PROGRAM MAIN
VAR
	//Required functions
	fbJson:FB_JsonSaxWriter;
	fbSaveFile :FB_SaveFile;
	fbReadJsonReal :FB_ReadJsonReal;
	
	//Triggers for testing
	bTrigger: BOOL:=TRUE;
	bSave:BOOL;
	bLoadJsonFile:BOOL;
	
	//Buffer required to save the information in the json file. If a huge value is required, then change the buffer size 
	sBuffer :STRING(255);
	
	//Random values for simulation
	r1:LREAL;
	r2:LREAL;
	r3:LREAL;
	r4:LREAL;
	dtTime: DATE_AND_TIME;

	//Variables to read the json file
	fSensor1Value :LREAL;
	fSensor2Value: LREAL;
	fSensor3Value: LREAL;
	fSensor4Value: LREAL;
	fTimeStampValue: LREAL;
	
END_VAR


//Trigger the following to gather random numbers
IF bTrigger THEN
	r1:=r1+(1.0/3.0);
	r2:=r2+(2.0/3.0);
	r3:=r3+(5.0/3.0);
	r4:=r4+(7.0/3.0);
	
	// JSON Object creation
	fbJson.StartObject(); //Open Bracket
		fbJson.AddKeyLreal('Sensor1',r1);
		fbJson.AddKeyLreal('Sensor2',r2);
		fbJson.AddKeyLreal('Sensor3',r3);
		fbJson.AddKeyLreal('Sensor4',r4);
		fbJson.AddKeyDateTime('TimeStamp',dtTime); //Extra data type to add some more info
	fbJson.EndObject(); //Close Bracket
	//Document creation
	sBuffer := fbJson.GetDocument();
	//Reset to get only one execution values
	fbJson.ResetDocument();
	
END_IF

//Save information, trigger bSave to create the file
IF bSave THEN
	fbSaveFile(sPath:='C:\TwinCAT\3.1\Boot\MyData.json',AmsNetId:='',pBuffer:=ADR(sBuffer), nBufLen:= LEN(sBuffer));
	IF fbSaveFile.SaveFileDone AND NOT fbSaveFile.ErrorSaveFile THEN
	bSave:=FALSE;
	END_IF
END_IF

//Test, trigger bLoadJsonFile to read the information
IF bLoadJsonFile THEN
	fbReadJsonReal(Member:='Sensor1',sPath:='C:\TwinCAT\3.1\Boot\MyData.json',fReadValue=>);
	fSensor1Value:= fbReadJsonReal.fReadValue;
	
	fbReadJsonReal(Member:='Sensor2',sPath:='C:\TwinCAT\3.1\Boot\MyData.json',fReadValue=>);
	fSensor2Value:= fbReadJsonReal.fReadValue;
	
	fbReadJsonReal(Member:='Sensor3',sPath:='C:\TwinCAT\3.1\Boot\MyData.json',fReadValue=>);
	fSensor3Value:= fbReadJsonReal.fReadValue;
	
	fbReadJsonReal(Member:='Sensor4',sPath:='C:\TwinCAT\3.1\Boot\MyData.json',fReadValue=>);
	fSensor4Value:= fbReadJsonReal.fReadValue;
	
	fbReadJsonReal(Member:='TimeStamp',sPath:='C:\TwinCAT\3.1\Boot\MyData.json',fReadValue=>);
	fTimeStampValue:= fbReadJsonReal.fReadValue;
END_IF

END_PROGRAM

(* stored: Version 1.1.0.1, ProductVersion 3.1.4024.14
   POU MAIN: Id {81fdac0f-1e0d-486a-ba31-7d84129b3f10}, SpecialFunc None *)
